// SIMATIC STEP 7 (V5.x) project ZEn01_07_STEP7__Dist_IO
// CPU: CPU315-2 DP
// station: Hardware
// station: SIMATIC 300(1)
// station: _S7H_BUSSYSTEM_CT
// program: S7-Program(1)

ORGANIZATION_BLOCK OB 1
VERSION : 0.1
VAR_TEMP
  OB1_EV_CLASS : BYTE ;	//Bits 0 to 3 = 1 (incoming event), bits 4 to 7 = 1 (event class 1)
  OB1_SCAN_1 : BYTE ;	//1 (cold restart scan 1 of OB1), 3 (scan 2-n of OB1)
  OB1_PRIORITY : BYTE ;	//1 (priority of 1 is lowest)
  OB1_OB_NUMBR : BYTE ;	//1 (organization block 1, OB1)
  OB1_RESERVED_1 : BYTE ;	//Reserved for system
  OB1_RESERVED_2 : BYTE ;	//Reserved for system
  OB1_PREV_CYCLE : INT ;	//Cycle time of previous OB1 scan (milliseconds)
  OB1_MIN_CYCLE : INT ;	//Minimum cycle time of OB1 (milliseconds)
  OB1_MAX_CYCLE : INT ;	//Maximum cycle time of OB1 (milliseconds)
  OB1_DATE_TIME : DATE_AND_TIME ;	//Date and time OB1 started
END_VAR
BEGIN
// (block stored without names or comments; labels and parameter names are numbered)
END_ORGANIZATION_BLOCK

ORGANIZATION_BLOCK OB 1
VERSION : 0.1
VAR_TEMP
  OB1_EV_CLASS : BYTE ;	//Bits 0 to 3 = 1 (incoming event), bits 4 to 7 = 1 (event class 1)
  OB1_SCAN_1 : BYTE ;	//1 (cold restart scan 1 of OB1), 3 (scan 2-n of OB1)
  OB1_PRIORITY : BYTE ;	//1 (priority of 1 is lowest)
  OB1_OB_NUMBR : BYTE ;	//1 (organization block 1, OB1)
  OB1_RESERVED_1 : BYTE ;	//Reserved for system
  OB1_RESERVED_2 : BYTE ;	//Reserved for system
  OB1_PREV_CYCLE : INT ;	//Cycle time of previous OB1 scan (milliseconds)
  OB1_MIN_CYCLE : INT ;	//Minimum cycle time of OB1 (milliseconds)
  OB1_MAX_CYCLE : INT ;	//Maximum cycle time of OB1 (milliseconds)
  OB1_DATE_TIME : DATE_AND_TIME ;	//Date and time OB1 started
END_VAR
BEGIN
// (block stored without names or comments; labels and parameter names are numbered)
END_ORGANIZATION_BLOCK
